{attribute 'qualified_only'}
{attribute 'strict'}
TYPE ST_LaudaActualValuesCollection :
STRUCT
	BathTemperature		: REAL;
	TemperatureSetpoint	: REAL;
	PumpStage			: UINT;
	StandBy				: BOOL;
	LiquidLevel			: UINT;
END_STRUCT
END_TYPE

(* stored: Version 1.1.0.1, ProductVersion 3.1.4024.13
   DUT ST_LaudaActualValuesCollection: Id {9d4a1ed1-cd3c-0e37-06cb-e1dfd2a22cbd} *)
